(* PLC project PLC411_DI, home PLC411_DI 1 *)
(* stored: creationDateTime 2023-04-11T09:37:45, productRelease 0, modificationDateTime 2023-04-11T13:46:01, version 1 *)

(* Установка режима работы дискретного входа *)
FUNCTION_BLOCK DIMode
  VAR_INPUT
    DIn : BYTE := 0;  (* номер входа *)
    M : BYTE := 0;  (* режим работы *)
  END_VAR
  VAR_OUTPUT
    Om : BYTE := 0;  (* режим работы (установленный) *)
    Ok : BYTE := 0;  (* код результата исполнения блока *)
  END_VAR

            {extern void App_DIMode(DIMODE*);App_DIMode(data__);}

          
END_FUNCTION_BLOCK

(* Получить значение нормального дискретного входа *)
FUNCTION_BLOCK DINorm
  VAR_INPUT
    DIn : BYTE := 0;  (* номер входа *)
  END_VAR
  VAR_OUTPUT
    Ov : BOOL := FALSE;  (* значение *)
    Ok : BYTE := 0;  (* код результата исполнения блока *)
  END_VAR

            {extern void App_DINorm(DINORM*);App_DINorm(data__);}

          
END_FUNCTION_BLOCK

(* Получить значение входа тахометра *)
FUNCTION_BLOCK DITach
  VAR_INPUT
    DIn : BYTE := 0;  (* номер входа *)
    Ref : WORD := 0;  (* уставка *)
    RefEn : BOOL := FALSE;  (* разрешение работы по уставке *)
  END_VAR
  VAR_OUTPUT
    Ov : WORD := 0;  (* значение *)
    Oref : BOOL := FALSE;  (* признак достижения уставки *)
    Ok : BYTE := 0;  (* код результата исполнения блока *)
  END_VAR

            {extern void App_DITach(DITACH*);App_DITach(data__);}

          
END_FUNCTION_BLOCK

(* Получить значение счетного входа *)
FUNCTION_BLOCK DICntr
  VAR_INPUT
    DIn : BYTE := 0;  (* номер входа *)
    Ref : DWORD := 0;  (* уставка *)
    RefEn : BOOL := FALSE;  (* разрешение работы по уставке *)
  END_VAR
  VAR_OUTPUT
    Ov : DWORD := 0;  (* значение счетчика *)
    Oref : BOOL := FALSE;  (* признак достижения уставки *)
    Ok : BYTE := 0;  (* код результата исполнения блока *)
  END_VAR

            {extern void App_DICntr(DICNTR*);App_DICntr(data__);}

          
END_FUNCTION_BLOCK

(* Сброс счетного входа *)
FUNCTION_BLOCK DICntrRst
  VAR_INPUT
    DIn : BYTE := 0;  (* номер входа *)
    Rst : BOOL := FALSE;  (* команда сброса *)
  END_VAR
  VAR_OUTPUT
    Ok : BYTE := 0;  (* код результата исполнения блока *)
  END_VAR

            {extern void App_DICntrRst(DICNTRRST*);App_DICntrRst(data__);}

          
END_FUNCTION_BLOCK

(* Получить значения входов счетного энкодера *)
FUNCTION_BLOCK DIEnc
  VAR_INPUT
    DIn : BYTE := 0;  (* номер первичного группового входа *)
    RefA : DWORD := 0;  (* уставка счетчика фазы A *)
    RefAEn : BOOL := FALSE;  (* разрешение работы счетчика фазы A по уставке *)
    RefB : DWORD := 0;  (* уставка счетчика фазы B *)
    RefBEn : BOOL := FALSE;  (* разрешение работы счетчика фазы B по уставке *)
    RefT : WORD := 0;  (* уставка тахометра *)
    RefTEn : BOOL := FALSE;  (* разрешение работы тахометра по уставке *)
  END_VAR
  VAR_OUTPUT
    OA : DWORD := 0;  (* значение счетчика фазы A *)
    OAref : BOOL := FALSE;  (* признак достижения уставки счетчиком фазы A *)
    OB : DWORD := 0;  (* значение счетчика фазы B *)
    OBref : BOOL := FALSE;  (* признак достижения уставки счетчиком фазы B *)
    OT : WORD := 0;  (* значение тахометра *)
    OTref : BOOL := FALSE;  (* признак достижения уставки тахометром *)
    Ok : BYTE := 0;  (* код результата исполнения блока *)
  END_VAR

            {extern void App_DIEnc(DIENC*);App_DIEnc(data__);}

          
END_FUNCTION_BLOCK
